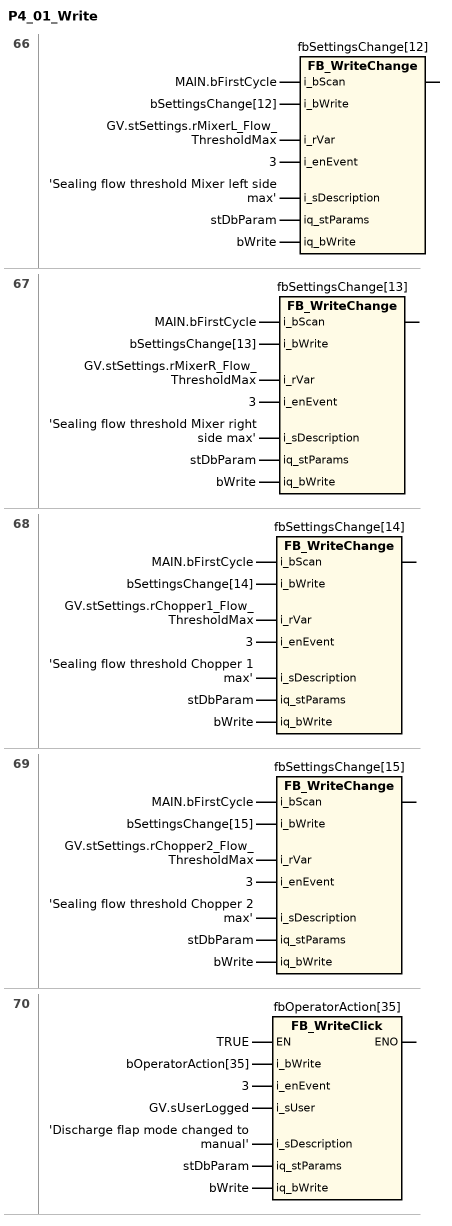
// NETWORK 66
fbSettingsChange[12](
    i_bScan := MAIN.bFirstCycle,
    i_bWrite := bSettingsChange[12],
    i_rVar := GV.stSettings.rMixerL_Flow_ThresholdMax,
    i_enEvent := 3,
    i_sDescription := 'Sealing flow threshold Mixer left side max',
    iq_stParams := stDbParam,
    iq_bWrite := bWrite); // FB_WriteChange

// NETWORK 67
fbSettingsChange[13](
    i_bScan := MAIN.bFirstCycle,
    i_bWrite := bSettingsChange[13],
    i_rVar := GV.stSettings.rMixerR_Flow_ThresholdMax,
    i_enEvent := 3,
    i_sDescription := 'Sealing flow threshold Mixer right side max',
    iq_stParams := stDbParam,
    iq_bWrite := bWrite); // FB_WriteChange

// NETWORK 68
fbSettingsChange[14](
    i_bScan := MAIN.bFirstCycle,
    i_bWrite := bSettingsChange[14],
    i_rVar := GV.stSettings.rChopper1_Flow_ThresholdMax,
    i_enEvent := 3,
    i_sDescription := 'Sealing flow threshold Chopper 1 max',
    iq_stParams := stDbParam,
    iq_bWrite := bWrite); // FB_WriteChange

// NETWORK 69
fbSettingsChange[15](
    i_bScan := MAIN.bFirstCycle,
    i_bWrite := bSettingsChange[15],
    i_rVar := GV.stSettings.rChopper2_Flow_ThresholdMax,
    i_enEvent := 3,
    i_sDescription := 'Sealing flow threshold Chopper 2 max',
    iq_stParams := stDbParam,
    iq_bWrite := bWrite); // FB_WriteChange

// NETWORK 70
fbOperatorAction[35](
    i_bWrite := bOperatorAction[35],
    i_enEvent := 3,
    i_sUser := GV.sUserLogged,
    i_sDescription := 'Discharge flap mode changed to manual',
    iq_stParams := stDbParam,
    iq_bWrite := bWrite); // FB_WriteClick

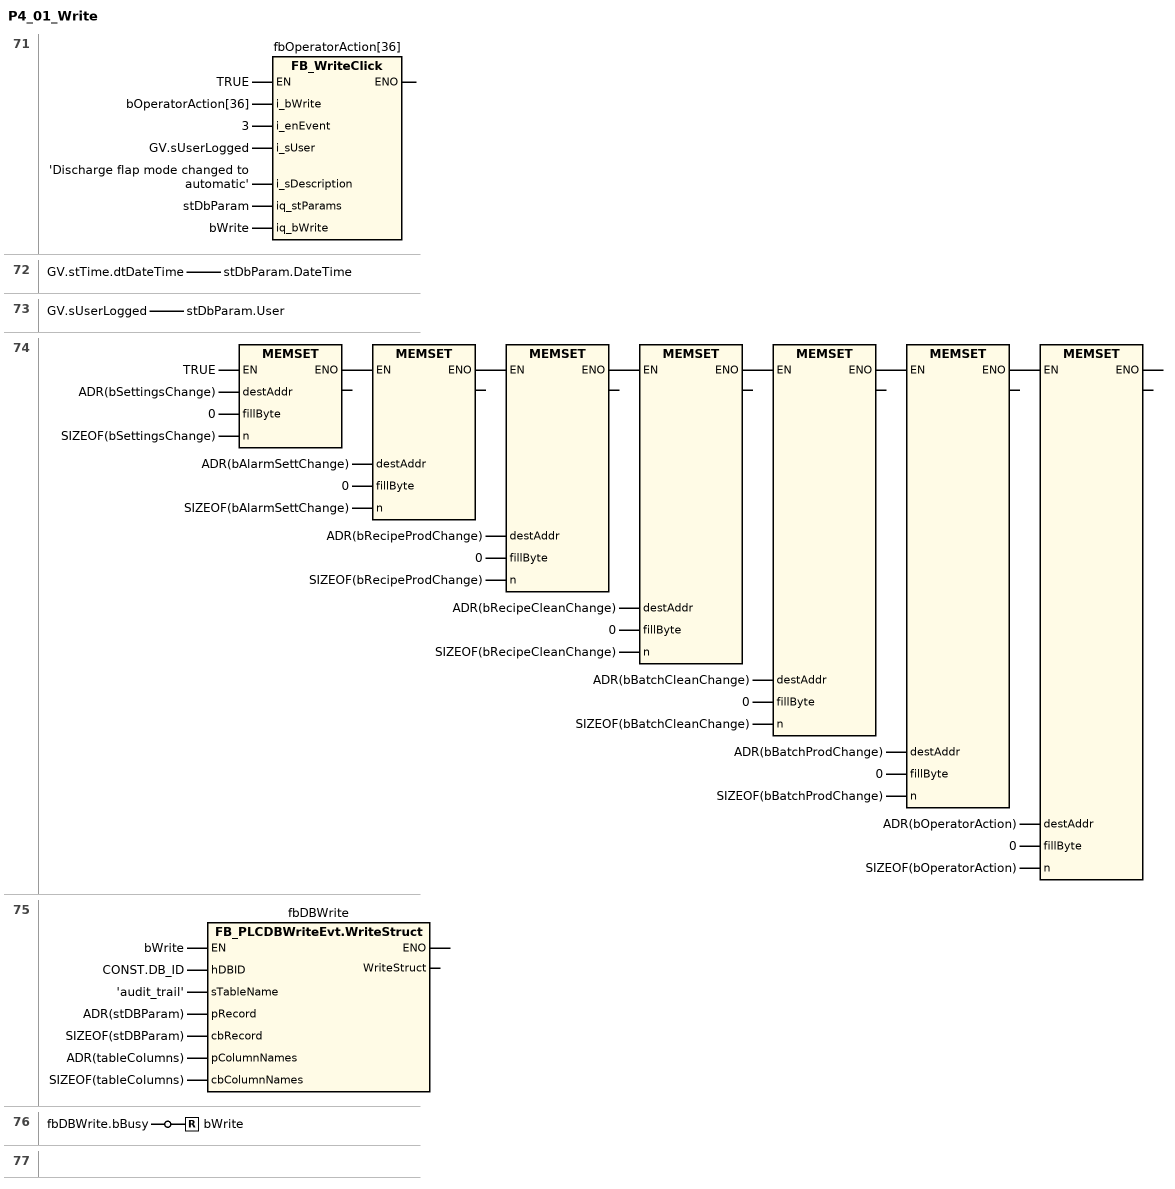
// NETWORK 71
fbOperatorAction[36](
    i_bWrite := bOperatorAction[36],
    i_enEvent := 3,
    i_sUser := GV.sUserLogged,
    i_sDescription := 'Discharge flap mode changed to automatic',
    iq_stParams := stDbParam,
    iq_bWrite := bWrite); // FB_WriteClick

// NETWORK 72
stDbParam.DateTime := GV.stTime.dtDateTime;

// NETWORK 73
stDbParam.User := GV.sUserLogged;

// NETWORK 74
MEMSET(destAddr := ADR(bSettingsChange), fillByte := 0, n := SIZEOF(bSettingsChange));
MEMSET(destAddr := ADR(bAlarmSettChange), fillByte := 0, n := SIZEOF(bAlarmSettChange));
MEMSET(destAddr := ADR(bRecipeProdChange), fillByte := 0, n := SIZEOF(bRecipeProdChange));
MEMSET(destAddr := ADR(bRecipeCleanChange), fillByte := 0, n := SIZEOF(bRecipeCleanChange));
MEMSET(destAddr := ADR(bBatchCleanChange), fillByte := 0, n := SIZEOF(bBatchCleanChange));
MEMSET(destAddr := ADR(bBatchProdChange), fillByte := 0, n := SIZEOF(bBatchProdChange));
MEMSET(destAddr := ADR(bOperatorAction), fillByte := 0, n := SIZEOF(bOperatorAction));

// NETWORK 75
IF bWrite THEN
    fbDBWrite.WriteStruct(
        hDBID := CONST.DB_ID,
        sTableName := 'audit_trail',
        pRecord := ADR(stDBParam),
        cbRecord := SIZEOF(stDBParam),
        pColumnNames := ADR(tableColumns),
        cbColumnNames := SIZEOF(tableColumns));
END_IF

// NETWORK 76
bWrite R= NOT fbDBWrite.bBusy;

// NETWORK 77

END_PROGRAM

// ---- FB/Database/FB_WriteChange.TcPOU
FUNCTION_BLOCK FB_WriteChange
VAR_INPUT
	i_bScan			:BOOL;
	i_bWrite		:BOOL;
	i_rVar			:REAL;
	i_enEvent		:EN_BatchEvents;
	i_sDescription	:STRING;
END_VAR
VAR
	iVarOld			:REAL;
	bVarOld			:BOOL;
	Trig			:R_TRIG;
	bScan			:BOOL;
	Scan			:R_TRIG;
	Scan_TON		:TON;
END_VAR
VAR_IN_OUT
	iq_stParams		:ST_AuditTrail;
	iq_bWrite		:BOOL;
END_VAR

IF i_bScan THEN
	bScan:=TRUE;
END_IF
Scan_TON(IN:=bScan,PT:=T#1S);
IF Scan_TON.Q THEN
	iVarOld:=i_rVar;
	bScan:=FALSE;
END_IF
Trig(CLK:=i_bWrite);
IF Trig.Q AND NOT bScan AND iVarOld <> i_rVar THEN
	iq_stParams.Event:=TO_STRING(i_enEvent);
	iq_stParams.Description := i_sDescription;
	iq_stParams.Oldvalue:=REAL_TO_STRING(iVarOld);
	iq_stParams.Newvalue:=REAL_TO_STRING(i_rVar);
	iVarOld:=i_rVar;
	iq_bWrite:=TRUE;
END_IF

END_FUNCTION_BLOCK

// ---- FB/Database/FB_WriteChange_STR.TcPOU
FUNCTION_BLOCK FB_WriteChange_STR
VAR_INPUT
	i_bScan			:BOOL;
	i_bWrite		:BOOL;
	i_sVar			:STRING;
	i_enEvent		:EN_BatchEvents;
	i_sDescription	:STRING;
END_VAR
VAR
	sVarOld			:STRING;
	bVarOld			:BOOL;
	Trig			:R_TRIG;
	bScan			:BOOL;
	Scan_TON		:TON;
END_VAR
VAR_IN_OUT
	iq_stParams		:ST_AuditTrail;
	iq_bWrite		:BOOL;
END_VAR

IF i_bScan THEN
	bScan:=TRUE;
END_IF
Scan_TON(IN:=bScan,PT:=T#1S);
IF Scan_TON.Q THEN
	sVarOld:=i_sVar;
	bScan:=FALSE;
END_IF
Trig(CLK:=i_bWrite);
IF Trig.Q AND NOT bScan THEN
	iq_stParams.Event:=TO_STRING(i_enEvent);
	iq_stParams.Description := i_sDescription;
	iq_stParams.Oldvalue:=sVarOld;
	iq_stParams.Newvalue:=i_sVar;
	sVarOld:=i_sVar;
	iq_bWrite:=TRUE;
END_IF

END_FUNCTION_BLOCK

// ---- FB/Database/FB_WriteClick.TcPOU
FUNCTION_BLOCK FB_WriteClick
VAR_INPUT
	i_bWrite		:BOOL;
	i_enEvent		:EN_BatchEvents;
	i_sUser			:STRING;
	i_sDescription	:STRING;
END_VAR
VAR
	Trig			:R_TRIG;
END_VAR
VAR_IN_OUT
	iq_stParams		:ST_AuditTrail;
	iq_bWrite		:BOOL;
END_VAR

(*Trig(CLK:=i_bWrite);
IF Trig.Q THEN
	iq_stParams.Event:=TO_STRING(i_enEvent);
	iq_stParams.Description := i_sDescription;
	iq_stParams.Oldvalue:='/';
	iq_stParams.Newvalue:='/';
	iq_bWrite:=TRUE;
END_IF
*)
IF i_bWrite THEN
	iq_stParams.Event:=TO_STRING(i_enEvent);
	iq_stParams.Description := i_sDescription;
	iq_stParams.Oldvalue:='/';
	iq_stParams.Newvalue:='/';
	iq_bWrite:=TRUE;
END_IF

END_FUNCTION_BLOCK

// ---- POUs/4. Audit Trail/P4_02_Read.TcPOU
PROGRAM P4_02_Read
VAR
	fbDBRead    	:FB_PLCDBCmdEvt(sNetID:=CONST.AMS_NETID, tTimeout:=DEFAULT_ADS_TIMEOUT);
	
	tableColumns	:ARRAY [0..5] OF STRING(50) := ['DateTime', 'User', 'Event', 'Description', 'OldValue', 'NewValue'];
	arrParam		:ARRAY [0..5] OF ST_ExpParameter := [(sParaName := 'DateTime', nParaSize := 4, eParaType := E_EXPPARAMETERTYPE.DateTime), 
														(sParaName := 'User', nParaSize := 101, eParaType := E_EXPPARAMETERTYPE.STRING_), 
														(sParaName := 'Event', nParaSize := 101, eParaType := E_EXPPARAMETERTYPE.STRING_), 
														(sParaName := 'Description', nParaSize := 101, eParaType := E_EXPPARAMETERTYPE.STRING_), 
														(sParaName := 'OldValue', nParaSize := 101, eParaType := E_EXPPARAMETERTYPE.STRING_), 
														(sParaName := 'NewValue', nParaSize := 101, eParaType := E_EXPPARAMETERTYPE.STRING_)];
	stRecord		:ARRAY[0..999] OF ST_AuditTrail;	
	
	stDBParam 		:ST_AuditTrail;	
	nRecords		:UDINT;
	sCmd			:STRING[300];

END_VAR
VAR // added by the converter: edge detectors and wires of the graphical bodies
    _w1 : BOOL;
END_VAR

//**************HMI FILTER - COMPOSE QUERY***************
sCmd:='SELECT * FROM `audit_trail`';
IF GV.stHMI.stAudit_Ctrl.bFilter THEN
	
	IF GV.stHMI.stAudit_Ctrl.enFilter_Event <> 0 THEN
		sCmd:=CONCAT(sCmd,'WHERE `Event` = $'');
		sCmd:=CONCAT(sCmD,TO_STRING(GV.stHMI.stAudit_Ctrl.enFilter_Event));
		sCmd:=CONCAT(sCmd,'$'');
	END_IF
	IF GV.stHMI.stAudit_Ctrl.sFilter_User <> GV.sEmptyString THEN
		IF GV.stHMI.stAudit_Ctrl.enFilter_Event = 0 THEN
			sCmd:=CONCAT(sCmd,'WHERE `User` LIKE $'%');
		ELSE
			sCmd:=CONCAT(sCmd,'AND `User` LIKE $'%');
		END_IF
		sCmd:=CONCAT(sCmD,GV.stHMI.stAudit_Ctrl.sFilter_User);
		sCmd:=CONCAT(sCmd,'$'');
	END_IF
	IF GV.stHMI.stAudit_Ctrl.sFilter_Key <> GV.sEmptyString THEN
		IF GV.stHMI.stAudit_Ctrl.enFilter_Event = 0 AND GV.stHMI.stAudit_Ctrl.sFilter_User = GV.sEmptyString THEN
			sCmd:=CONCAT(sCmd,'WHERE `Description` LIKE $'%');
		ELSE
			sCmd:=CONCAT(sCmd,'AND `Description` LIKE $'%');
		END_IF
		sCmd:=CONCAT(sCmD,GV.stHMI.stAudit_Ctrl.sFilter_Key);
		sCmd:=CONCAT(sCmd,'%$'');
	END_IF
	IF GV.stHMI.stAudit_Ctrl.dtFilter_From <> GV.stHMI.stAudit_Ctrl.dtFilter_To THEN
		IF GV.stHMI.stAudit_Ctrl.enFilter_Event = 0 AND GV.stHMI.stAudit_Ctrl.sFilter_User = GV.sEmptyString AND GV.stHMI.stAudit_Ctrl.sFilter_Key = GV.sEmptyString THEN
				sCmd:=CONCAT(sCmd,'WHERE `DateTime` BETWEEN $'');
			ELSE
				sCmd:=CONCAT(sCmd,'AND `DateTime` BETWEEN $'');
			END_IF
			sCmd:=CONCAT(sCmd,RIGHT(DT_TO_STRING(GV.stHMI.stAudit_Ctrl.dtFilter_From),19));
			sCmd:=CONCAT(sCmd,'$' AND $'');
			sCmd:=CONCAT(sCmd,RIGHT(DT_TO_STRING(GV.stHMI.stAudit_Ctrl.dtFilter_To),19));
			sCmd:=CONCAT(sCmd,'$'');
	END_IF
	GV.stTX_Python.sAuditExportQuery:=sCmd;
END_IF
sCmd:=CONCAT(sCmd,' ORDER BY `DateTime` DESC');


ACT_Cmd();

ACTION ACT_Cmd:
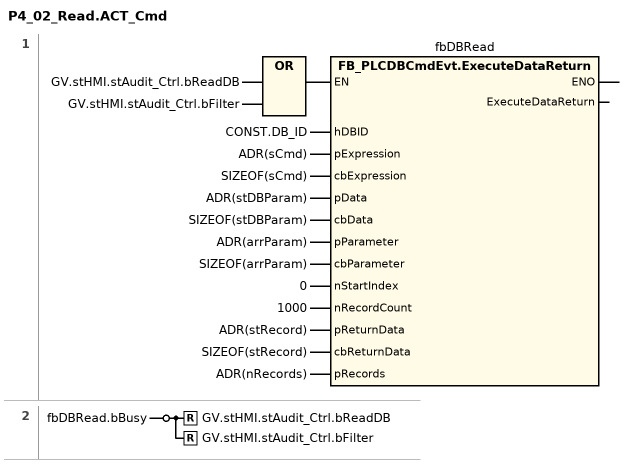
// NETWORK 1
IF GV.stHMI.stAudit_Ctrl.bReadDB OR GV.stHMI.stAudit_Ctrl.bFilter THEN
    fbDBRead.ExecuteDataReturn(
        hDBID := CONST.DB_ID,
        pExpression := ADR(sCmd),
        cbExpression := SIZEOF(sCmd),
        pData := ADR(stDBParam),
        cbData := SIZEOF(stDBParam),
        pParameter := ADR(arrParam),
        cbParameter := SIZEOF(arrParam),
        nStartIndex := 0,
        nRecordCount := 1000,
        pReturnData := ADR(stRecord),
        cbReturnData := SIZEOF(stRecord),
        pRecords := ADR(nRecords));
END_IF

// NETWORK 2
_w1 := NOT fbDBRead.bBusy;
GV.stHMI.stAudit_Ctrl.bReadDB R= _w1;
GV.stHMI.stAudit_Ctrl.bFilter R= _w1;
END_ACTION

END_PROGRAM

// ---- POUs/4. Audit Trail/P4_03_Export.TcPOU
PROGRAM P4_03_Export
VAR
	fbExportAudit					:FB_PythonScript;
END_VAR

VAR PERSISTENT
	sLastExportedAuditTime			:STRING;
	sLastExportedAuditName			:STRING;
END_VAR
VAR // added by the converter: edge detectors and wires of the graphical bodies
    _rt1, _rt2 : R_TRIG;
END_VAR

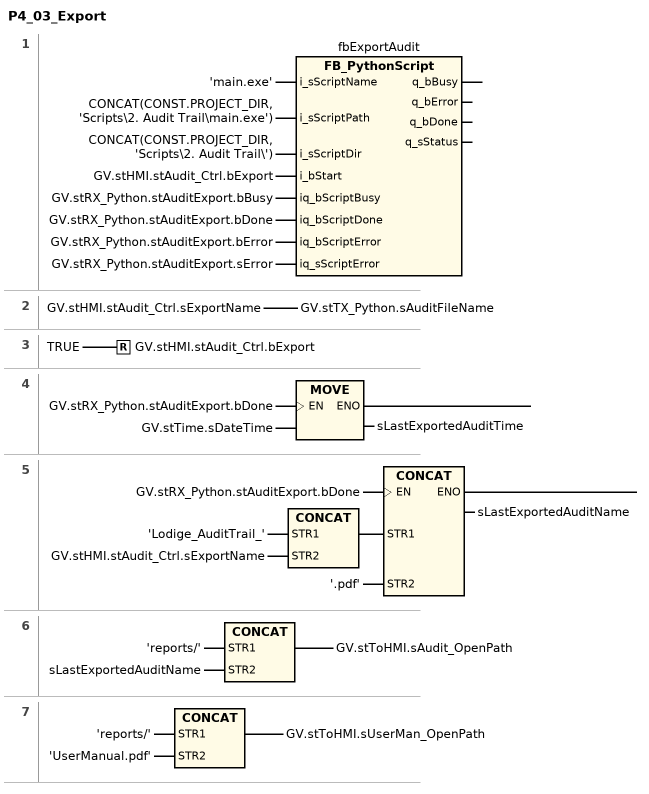
// NETWORK 1
fbExportAudit(
    i_sScriptName := 'main.exe',
    i_sScriptPath := CONCAT(CONST.PROJECT_DIR,'Scripts\2. Audit Trail\main.exe'),
    i_sScriptDir := CONCAT(CONST.PROJECT_DIR,'Scripts\2. Audit Trail\'),
    i_bStart := GV.stHMI.stAudit_Ctrl.bExport,
    iq_bScriptBusy := GV.stRX_Python.stAuditExport.bBusy,
    iq_bScriptDone := GV.stRX_Python.stAuditExport.bDone,
    iq_bScriptError := GV.stRX_Python.stAuditExport.bError,
    iq_sScriptError := GV.stRX_Python.stAuditExport.sError); // FB_PythonScript

// NETWORK 2
GV.stTX_Python.sAuditFileName := GV.stHMI.stAudit_Ctrl.sExportName;

// NETWORK 3
GV.stHMI.stAudit_Ctrl.bExport R= TRUE;

// NETWORK 4
_rt1(CLK := GV.stRX_Python.stAuditExport.bDone);
IF _rt1.Q THEN sLastExportedAuditTime := GV.stTime.sDateTime; END_IF

// NETWORK 5
_rt2(CLK := GV.stRX_Python.stAuditExport.bDone);
IF _rt2.Q THEN
    sLastExportedAuditName := CONCAT(STR1 := CONCAT(STR1 := 'Lodige_AuditTrail_', STR2 := GV.stHMI.stAudit_Ctrl.sExportName), STR2 := '.pdf');
END_IF

// NETWORK 6
GV.stToHMI.sAudit_OpenPath := CONCAT(STR1 := 'reports/', STR2 := sLastExportedAuditName);

// NETWORK 7
GV.stToHMI.sUserMan_OpenPath := CONCAT(STR1 := 'reports/', STR2 := 'UserManual.pdf');

END_PROGRAM

// ---- POUs/4. Audit Trail/P4_04_Delete.TcPOU
PROGRAM P4_04_Delete
VAR
	fbPLCDBCmd    	:FB_PLCDBCmdEvt(sNetID:=CONST.AMS_NETID, tTimeout:=DEFAULT_ADS_TIMEOUT);
	sCmdDelete		:STRING[80];
	
	arrParam		:ARRAY [0..5] OF ST_ExpParameter := [(sParaName := 'DateTime', nParaSize := 4, eParaType := E_EXPPARAMETERTYPE.DateTime), 
														(sParaName := 'User', nParaSize := 101, eParaType := E_EXPPARAMETERTYPE.STRING_), 
														(sParaName := 'Event', nParaSize := 101, eParaType := E_EXPPARAMETERTYPE.STRING_), 
														(sParaName := 'Description', nParaSize := 101, eParaType := E_EXPPARAMETERTYPE.STRING_), 
														(sParaName := 'OldValue', nParaSize := 101, eParaType := E_EXPPARAMETERTYPE.STRING_), 
														(sParaName := 'NewValue', nParaSize := 101, eParaType := E_EXPPARAMETERTYPE.STRING_)];
	
	stDBParam 		:ST_AuditTrail;	
END_VAR

sCmdDelete:='DELETE FROM `audit_trail`';
ACT_Cmd();

ACTION ACT_Cmd:
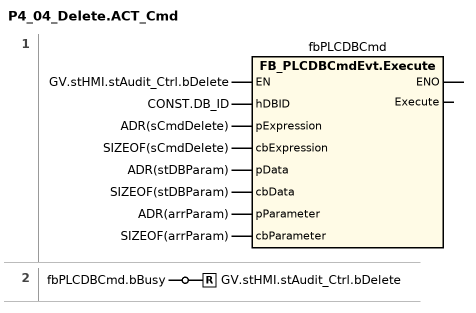
// NETWORK 1
IF GV.stHMI.stAudit_Ctrl.bDelete THEN
    fbPLCDBCmd.Execute(
        hDBID := CONST.DB_ID,
        pExpression := ADR(sCmdDelete),
        cbExpression := SIZEOF(sCmdDelete),
        pData := ADR(stDBParam),
        cbData := SIZEOF(stDBParam),
        pParameter := ADR(arrParam),
        cbParameter := SIZEOF(arrParam));
END_IF

// NETWORK 2
GV.stHMI.stAudit_Ctrl.bDelete R= NOT fbPLCDBCmd.bBusy;
END_ACTION

END_PROGRAM

// ---- POUs/4. Audit Trail/P4_05_Send.TcPOU
PROGRAM P4_05_Send
VAR
	fbAuditSend							:FB_PythonScript;
END_VAR
VAR // added by the converter: edge detectors and wires of the graphical bodies
    _rt1 : R_TRIG;
END_VAR

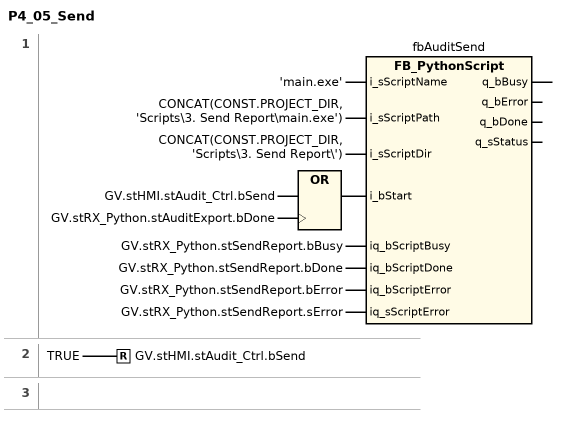
// NETWORK 1
_rt1(CLK := GV.stRX_Python.stAuditExport.bDone);
fbAuditSend(
    i_sScriptName := 'main.exe',
    i_sScriptPath := CONCAT(CONST.PROJECT_DIR,'Scripts\3. Send Report\main.exe'),
    i_sScriptDir := CONCAT(CONST.PROJECT_DIR,'Scripts\3. Send Report\'),
    i_bStart := GV.stHMI.stAudit_Ctrl.bSend OR _rt1.Q,
    iq_bScriptBusy := GV.stRX_Python.stSendReport.bBusy,
    iq_bScriptDone := GV.stRX_Python.stSendReport.bDone,
    iq_bScriptError := GV.stRX_Python.stSendReport.bError,
    iq_sScriptError := GV.stRX_Python.stSendReport.sError); // FB_PythonScript

// NETWORK 2
GV.stHMI.stAudit_Ctrl.bSend R= TRUE;

// NETWORK 3

END_PROGRAM

// ---- POUs/4. Audit Trail/P4_05_DIskSize.TcPOU
PROGRAM P4_05_DIskSize
VAR
	fbSize				:FB_PythonScript;
END_VAR

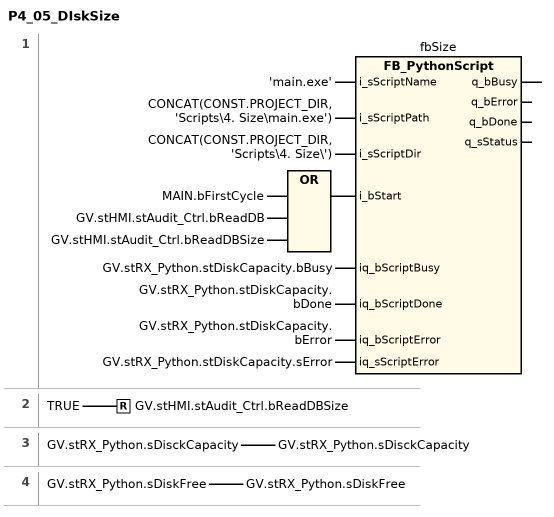
// NETWORK 1
fbSize(
    i_sScriptName := 'main.exe',
    i_sScriptPath := CONCAT(CONST.PROJECT_DIR,'Scripts\4. Size\main.exe'),
    i_sScriptDir := CONCAT(CONST.PROJECT_DIR,'Scripts\4. Size\'),
    i_bStart := MAIN.bFirstCycle OR GV.stHMI.stAudit_Ctrl.bReadDB OR GV.stHMI.stAudit_Ctrl.bReadDBSize,
    iq_bScriptBusy := GV.stRX_Python.stDiskCapacity.bBusy,
    iq_bScriptDone := GV.stRX_Python.stDiskCapacity.bDone,
    iq_bScriptError := GV.stRX_Python.stDiskCapacity.bError,
    iq_sScriptError := GV.stRX_Python.stDiskCapacity.sError); // FB_PythonScript

// NETWORK 2
GV.stHMI.stAudit_Ctrl.bReadDBSize R= TRUE;

// NETWORK 3
GV.stRX_Python.sDisckCapacity := GV.stRX_Python.sDisckCapacity;

// NETWORK 4
GV.stRX_Python.sDiskFree := GV.stRX_Python.sDiskFree;

END_PROGRAM

// ---- POUs/5. HMI/P5_00_MAIN.TcPOU
PROGRAM P5_00_MAIN
VAR

END_VAR

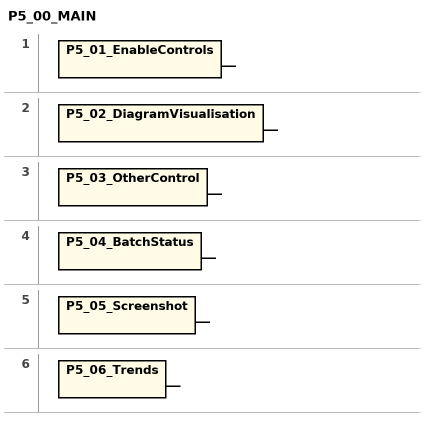
// NETWORK 1
P5_01_EnableControls();

// NETWORK 2
P5_02_DiagramVisualisation();

// NETWORK 3
P5_03_OtherControl();

// NETWORK 4
P5_04_BatchStatus();

// NETWORK 5
P5_05_Screenshot();

// NETWORK 6
P5_06_Trends();

END_PROGRAM

// ---- POUs/5. HMI/P5_01_EnableControls.TcPOU
PROGRAM P5_01_EnableControls
VAR
	tonDisableNext			:TON;
	tonDisablePrev			:TON;
END_VAR
VAR // added by the converter: edge detectors and wires of the graphical bodies
    _w1, _w2 : BOOL;
END_VAR

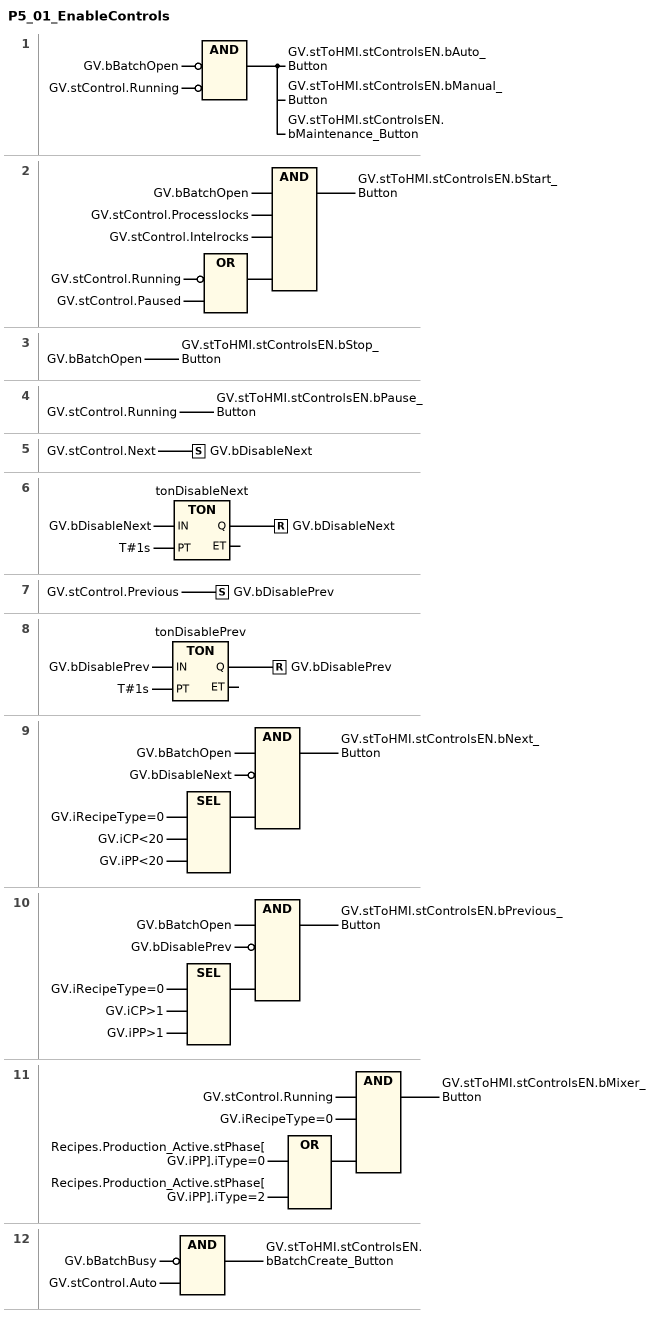
// NETWORK 1
_w1 := NOT GV.bBatchOpen AND NOT GV.stControl.Running;
GV.stToHMI.stControlsEN.bAuto_Button := _w1;
GV.stToHMI.stControlsEN.bManual_Button := _w1;
GV.stToHMI.stControlsEN.bMaintenance_Button := _w1;

// NETWORK 2
GV.stToHMI.stControlsEN.bStart_Button := GV.bBatchOpen AND GV.stControl.Processlocks AND GV.stControl.Intelrocks AND (NOT GV.stControl.Running OR GV.stControl.Paused);

// NETWORK 3
GV.stToHMI.stControlsEN.bStop_Button := GV.bBatchOpen;

// NETWORK 4
GV.stToHMI.stControlsEN.bPause_Button := GV.stControl.Running;

// NETWORK 5
GV.bDisableNext S= GV.stControl.Next;

// NETWORK 6
tonDisableNext(IN := GV.bDisableNext, PT := T#1s); // TON
GV.bDisableNext R= tonDisableNext.Q;

// NETWORK 7
GV.bDisablePrev S= GV.stControl.Previous;

// NETWORK 8
tonDisablePrev(IN := GV.bDisablePrev, PT := T#1s); // TON
GV.bDisablePrev R= tonDisablePrev.Q;

// NETWORK 9
GV.stToHMI.stControlsEN.bNext_Button := GV.bBatchOpen AND NOT GV.bDisableNext AND SEL(GV.iRecipeType=0, GV.iCP<20, GV.iPP<20);

// NETWORK 10
GV.stToHMI.stControlsEN.bPrevious_Button := GV.bBatchOpen AND NOT GV.bDisablePrev AND SEL(GV.iRecipeType=0, GV.iCP>1, GV.iPP>1);

// NETWORK 11
GV.stToHMI.stControlsEN.bMixer_Button := GV.stControl.Running AND (GV.iRecipeType=0) AND ((Recipes.Production_Active.stPhase[GV.iPP].iType=0) OR (Recipes.Production_Active.stPhase[GV.iPP].iType=2));

// NETWORK 12
GV.stToHMI.stControlsEN.bBatchCreate_Button := NOT GV.bBatchBusy AND GV.stControl.Auto;

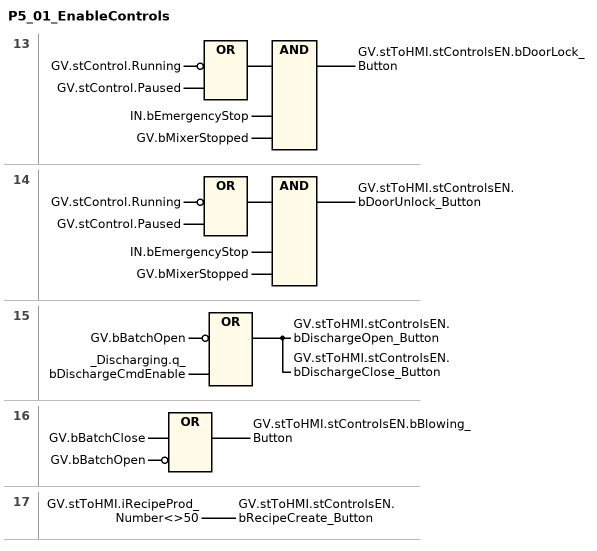
// NETWORK 13
GV.stToHMI.stControlsEN.bDoorLock_Button := (NOT GV.stControl.Running OR GV.stControl.Paused) AND IN.bEmergencyStop AND GV.bMixerStopped;

// NETWORK 14
GV.stToHMI.stControlsEN.bDoorUnlock_Button := (NOT GV.stControl.Running OR GV.stControl.Paused) AND IN.bEmergencyStop AND GV.bMixerStopped;

// NETWORK 15
_w2 := NOT GV.bBatchOpen OR _Discharging.q_bDischargeCmdEnable;
GV.stToHMI.stControlsEN.bDischargeOpen_Button := _w2;
GV.stToHMI.stControlsEN.bDischargeClose_Button := _w2;

// NETWORK 16
GV.stToHMI.stControlsEN.bBlowing_Button := GV.bBatchClose OR NOT GV.bBatchOpen;

// NETWORK 17
GV.stToHMI.stControlsEN.bRecipeCreate_Button := GV.stToHMI.iRecipeProd_Number<>50;

END_PROGRAM

// ---- POUs/5. HMI/P5_02_DiagramVisualisation.TcPOU
PROGRAM P5_02_DiagramVisualisation
VAR
END_VAR

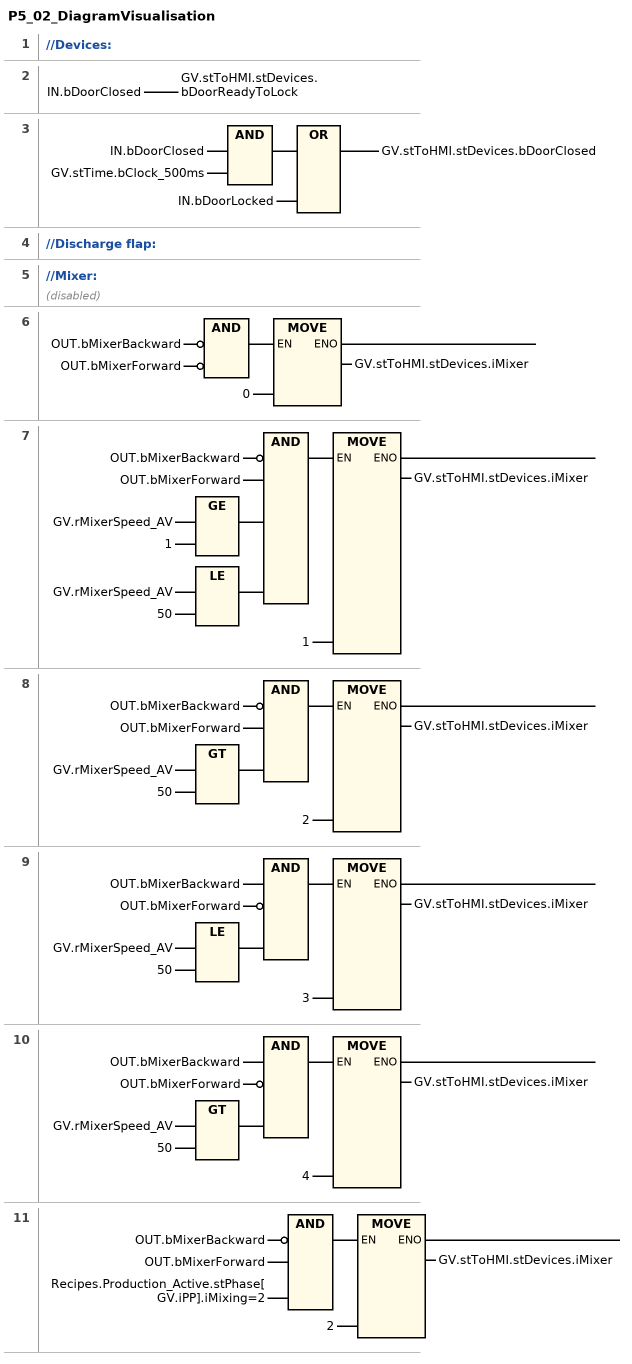
// NETWORK 1
// label: //Devices

// NETWORK 2
GV.stToHMI.stDevices.bDoorReadyToLock := IN.bDoorClosed;

// NETWORK 3
GV.stToHMI.stDevices.bDoorClosed := IN.bDoorClosed AND GV.stTime.bClock_500ms OR IN.bDoorLocked;

// NETWORK 4
// label: //Discharge flap

// NETWORK 5 (disabled)
// label: //Mixer

// NETWORK 6
IF NOT OUT.bMixerBackward AND NOT OUT.bMixerForward THEN GV.stToHMI.stDevices.iMixer := 0; END_IF

// NETWORK 7
IF NOT OUT.bMixerBackward AND OUT.bMixerForward AND GV.rMixerSpeed_AV >= 1 AND GV.rMixerSpeed_AV <= 50 THEN
    GV.stToHMI.stDevices.iMixer := 1;
END_IF

// NETWORK 8
IF NOT OUT.bMixerBackward AND OUT.bMixerForward AND GV.rMixerSpeed_AV > 50 THEN
    GV.stToHMI.stDevices.iMixer := 2;
END_IF

// NETWORK 9
IF OUT.bMixerBackward AND NOT OUT.bMixerForward AND GV.rMixerSpeed_AV <= 50 THEN
    GV.stToHMI.stDevices.iMixer := 3;
END_IF

// NETWORK 10
IF OUT.bMixerBackward AND NOT OUT.bMixerForward AND GV.rMixerSpeed_AV > 50 THEN
    GV.stToHMI.stDevices.iMixer := 4;
END_IF

// NETWORK 11
IF NOT OUT.bMixerBackward AND OUT.bMixerForward AND (Recipes.Production_Active.stPhase[GV.iPP].iMixing=2) THEN
    GV.stToHMI.stDevices.iMixer := 2;
END_IF

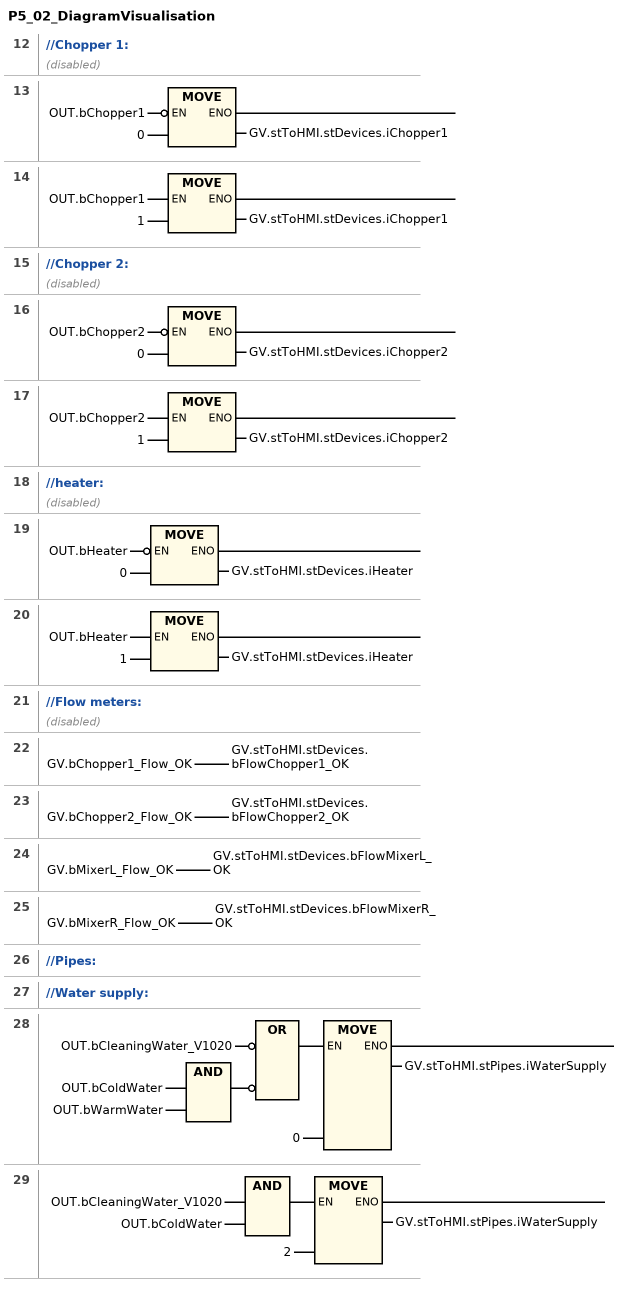
// NETWORK 12 (disabled)
// label: //Chopper 1

// NETWORK 13
IF NOT OUT.bChopper1 THEN GV.stToHMI.stDevices.iChopper1 := 0; END_IF

// NETWORK 14
IF OUT.bChopper1 THEN GV.stToHMI.stDevices.iChopper1 := 1; END_IF

// NETWORK 15 (disabled)
// label: //Chopper 2

// NETWORK 16
IF NOT OUT.bChopper2 THEN GV.stToHMI.stDevices.iChopper2 := 0; END_IF

// NETWORK 17
IF OUT.bChopper2 THEN GV.stToHMI.stDevices.iChopper2 := 1; END_IF

// NETWORK 18 (disabled)
// label: //heater

// NETWORK 19
IF NOT OUT.bHeater THEN GV.stToHMI.stDevices.iHeater := 0; END_IF

// NETWORK 20
IF OUT.bHeater THEN GV.stToHMI.stDevices.iHeater := 1; END_IF

// NETWORK 21 (disabled)
// label: //Flow meters

// NETWORK 22
GV.stToHMI.stDevices.bFlowChopper1_OK := GV.bChopper1_Flow_OK;

// NETWORK 23
GV.stToHMI.stDevices.bFlowChopper2_OK := GV.bChopper2_Flow_OK;

// NETWORK 24
GV.stToHMI.stDevices.bFlowMixerL_OK := GV.bMixerL_Flow_OK;

// NETWORK 25
GV.stToHMI.stDevices.bFlowMixerR_OK := GV.bMixerR_Flow_OK;

// NETWORK 26
// label: //Pipes

// NETWORK 27
// label: //Water supply

// NETWORK 28
IF NOT OUT.bCleaningWater_V1020 OR NOT (OUT.bColdWater AND OUT.bWarmWater) THEN
    GV.stToHMI.stPipes.iWaterSupply := 0;
END_IF

// NETWORK 29
IF OUT.bCleaningWater_V1020 AND OUT.bColdWater THEN GV.stToHMI.stPipes.iWaterSupply := 2; END_IF

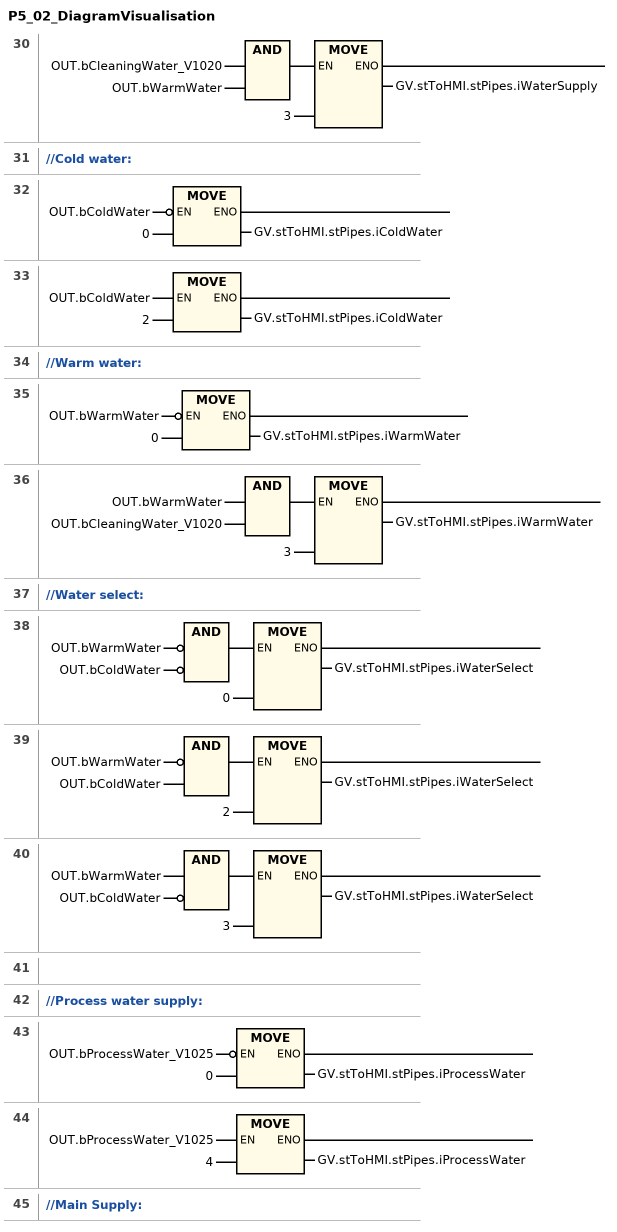
// NETWORK 30
IF OUT.bCleaningWater_V1020 AND OUT.bWarmWater THEN GV.stToHMI.stPipes.iWaterSupply := 3; END_IF

// NETWORK 31
// label: //Cold water

// NETWORK 32
IF NOT OUT.bColdWater THEN GV.stToHMI.stPipes.iColdWater := 0; END_IF

// NETWORK 33
IF OUT.bColdWater THEN GV.stToHMI.stPipes.iColdWater := 2; END_IF

// NETWORK 34
// label: //Warm water

// NETWORK 35
IF NOT OUT.bWarmWater THEN GV.stToHMI.stPipes.iWarmWater := 0; END_IF

// NETWORK 36
IF OUT.bWarmWater AND OUT.bCleaningWater_V1020 THEN GV.stToHMI.stPipes.iWarmWater := 3; END_IF

// NETWORK 37
// label: //Water select

// NETWORK 38
IF NOT OUT.bWarmWater AND NOT OUT.bColdWater THEN GV.stToHMI.stPipes.iWaterSelect := 0; END_IF

// NETWORK 39
IF NOT OUT.bWarmWater AND OUT.bColdWater THEN GV.stToHMI.stPipes.iWaterSelect := 2; END_IF

// NETWORK 40
IF OUT.bWarmWater AND NOT OUT.bColdWater THEN GV.stToHMI.stPipes.iWaterSelect := 3; END_IF

// NETWORK 41

// NETWORK 42
// label: //Process water supply

// NETWORK 43
IF NOT OUT.bProcessWater_V1025 THEN GV.stToHMI.stPipes.iProcessWater := 0; END_IF

// NETWORK 44
IF OUT.bProcessWater_V1025 THEN GV.stToHMI.stPipes.iProcessWater := 4; END_IF

// NETWORK 45
// label: //Main Supply

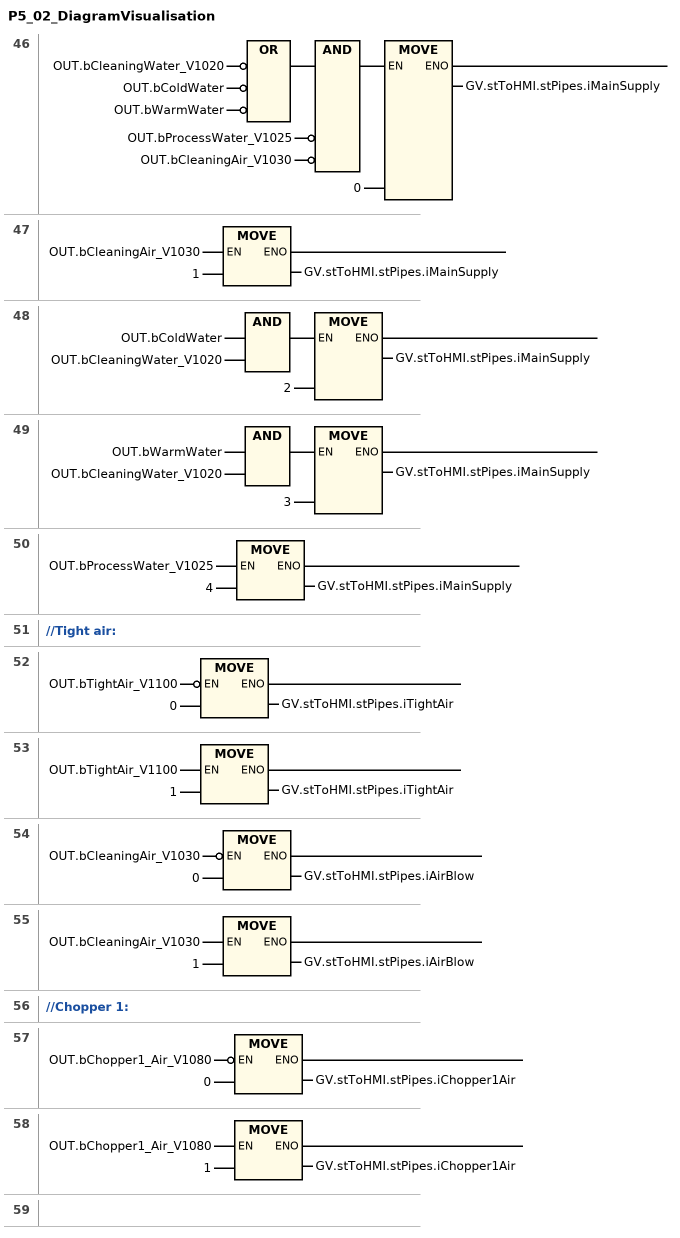
// NETWORK 46
IF (NOT OUT.bCleaningWater_V1020 OR NOT OUT.bColdWater OR NOT OUT.bWarmWater) AND NOT OUT.bProcessWater_V1025 AND NOT OUT.bCleaningAir_V1030 THEN
    GV.stToHMI.stPipes.iMainSupply := 0;
END_IF

// NETWORK 47
IF OUT.bCleaningAir_V1030 THEN GV.stToHMI.stPipes.iMainSupply := 1; END_IF

// NETWORK 48
IF OUT.bColdWater AND OUT.bCleaningWater_V1020 THEN GV.stToHMI.stPipes.iMainSupply := 2; END_IF

// NETWORK 49
IF OUT.bWarmWater AND OUT.bCleaningWater_V1020 THEN GV.stToHMI.stPipes.iMainSupply := 3; END_IF

// NETWORK 50
IF OUT.bProcessWater_V1025 THEN GV.stToHMI.stPipes.iMainSupply := 4; END_IF

// NETWORK 51
// label: //Tight air

// NETWORK 52
IF NOT OUT.bTightAir_V1100 THEN GV.stToHMI.stPipes.iTightAir := 0; END_IF

// NETWORK 53
IF OUT.bTightAir_V1100 THEN GV.stToHMI.stPipes.iTightAir := 1; END_IF

// NETWORK 54
IF NOT OUT.bCleaningAir_V1030 THEN GV.stToHMI.stPipes.iAirBlow := 0; END_IF

// NETWORK 55
IF OUT.bCleaningAir_V1030 THEN GV.stToHMI.stPipes.iAirBlow := 1; END_IF

// NETWORK 56
// label: //Chopper 1

// NETWORK 57
IF NOT OUT.bChopper1_Air_V1080 THEN GV.stToHMI.stPipes.iChopper1Air := 0; END_IF

// NETWORK 58
IF OUT.bChopper1_Air_V1080 THEN GV.stToHMI.stPipes.iChopper1Air := 1; END_IF

// NETWORK 59

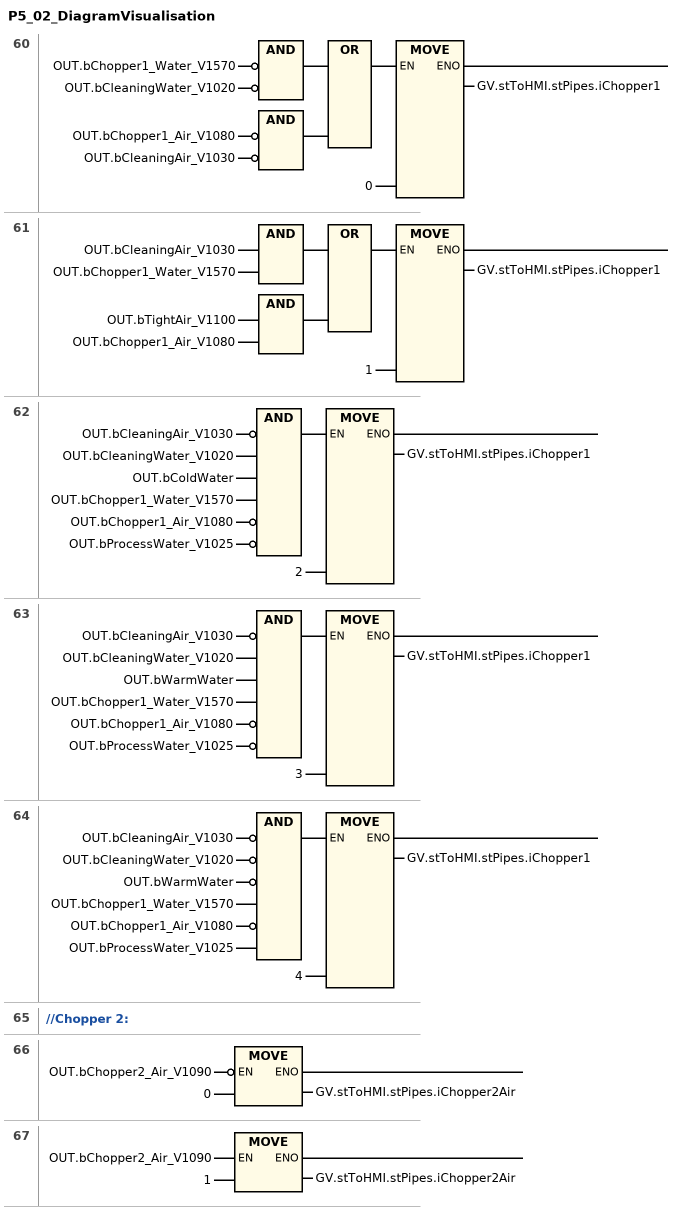
// NETWORK 60
IF NOT OUT.bChopper1_Water_V1570 AND NOT OUT.bCleaningWater_V1020 OR NOT OUT.bChopper1_Air_V1080 AND NOT OUT.bCleaningAir_V1030 THEN
    GV.stToHMI.stPipes.iChopper1 := 0;
END_IF

// NETWORK 61
IF OUT.bCleaningAir_V1030 AND OUT.bChopper1_Water_V1570 OR OUT.bTightAir_V1100 AND OUT.bChopper1_Air_V1080 THEN
    GV.stToHMI.stPipes.iChopper1 := 1;
END_IF

// NETWORK 62
IF NOT OUT.bCleaningAir_V1030 AND OUT.bCleaningWater_V1020 AND OUT.bColdWater AND OUT.bChopper1_Water_V1570 AND NOT OUT.bChopper1_Air_V1080 AND NOT OUT.bProcessWater_V1025 THEN
    GV.stToHMI.stPipes.iChopper1 := 2;
END_IF

// NETWORK 63
IF NOT OUT.bCleaningAir_V1030 AND OUT.bCleaningWater_V1020 AND OUT.bWarmWater AND OUT.bChopper1_Water_V1570 AND NOT OUT.bChopper1_Air_V1080 AND NOT OUT.bProcessWater_V1025 THEN
    GV.stToHMI.stPipes.iChopper1 := 3;
END_IF

// NETWORK 64
IF NOT OUT.bCleaningAir_V1030 AND NOT OUT.bCleaningWater_V1020 AND NOT OUT.bWarmWater AND OUT.bChopper1_Water_V1570 AND NOT OUT.bChopper1_Air_V1080 AND OUT.bProcessWater_V1025 THEN
    GV.stToHMI.stPipes.iChopper1 := 4;
END_IF

// NETWORK 65
// label: //Chopper 2

// NETWORK 66
IF NOT OUT.bChopper2_Air_V1090 THEN GV.stToHMI.stPipes.iChopper2Air := 0; END_IF

// NETWORK 67
IF OUT.bChopper2_Air_V1090 THEN GV.stToHMI.stPipes.iChopper2Air := 1; END_IF

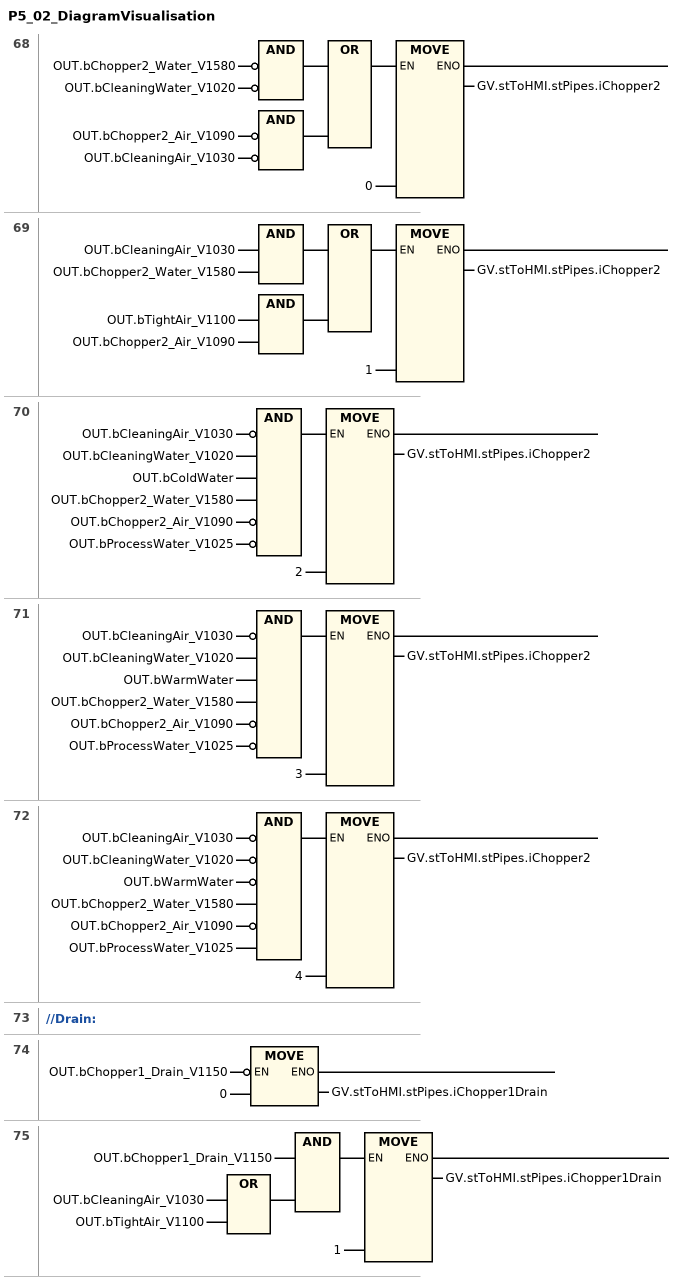
// NETWORK 68
IF NOT OUT.bChopper2_Water_V1580 AND NOT OUT.bCleaningWater_V1020 OR NOT OUT.bChopper2_Air_V1090 AND NOT OUT.bCleaningAir_V1030 THEN
    GV.stToHMI.stPipes.iChopper2 := 0;
END_IF

// NETWORK 69
IF OUT.bCleaningAir_V1030 AND OUT.bChopper2_Water_V1580 OR OUT.bTightAir_V1100 AND OUT.bChopper2_Air_V1090 THEN
    GV.stToHMI.stPipes.iChopper2 := 1;
END_IF

// NETWORK 70
IF NOT OUT.bCleaningAir_V1030 AND OUT.bCleaningWater_V1020 AND OUT.bColdWater AND OUT.bChopper2_Water_V1580 AND NOT OUT.bChopper2_Air_V1090 AND NOT OUT.bProcessWater_V1025 THEN
    GV.stToHMI.stPipes.iChopper2 := 2;
END_IF

// NETWORK 71
IF NOT OUT.bCleaningAir_V1030 AND OUT.bCleaningWater_V1020 AND OUT.bWarmWater AND OUT.bChopper2_Water_V1580 AND NOT OUT.bChopper2_Air_V1090 AND NOT OUT.bProcessWater_V1025 THEN
    GV.stToHMI.stPipes.iChopper2 := 3;
END_IF

// NETWORK 72
IF NOT OUT.bCleaningAir_V1030 AND NOT OUT.bCleaningWater_V1020 AND NOT OUT.bWarmWater AND OUT.bChopper2_Water_V1580 AND NOT OUT.bChopper2_Air_V1090 AND OUT.bProcessWater_V1025 THEN
    GV.stToHMI.stPipes.iChopper2 := 4;
END_IF

// NETWORK 73
// label: //Drain

// NETWORK 74
IF NOT OUT.bChopper1_Drain_V1150 THEN GV.stToHMI.stPipes.iChopper1Drain := 0; END_IF

// NETWORK 75
IF OUT.bChopper1_Drain_V1150 AND (OUT.bCleaningAir_V1030 OR OUT.bTightAir_V1100) THEN
    GV.stToHMI.stPipes.iChopper1Drain := 1;
END_IF

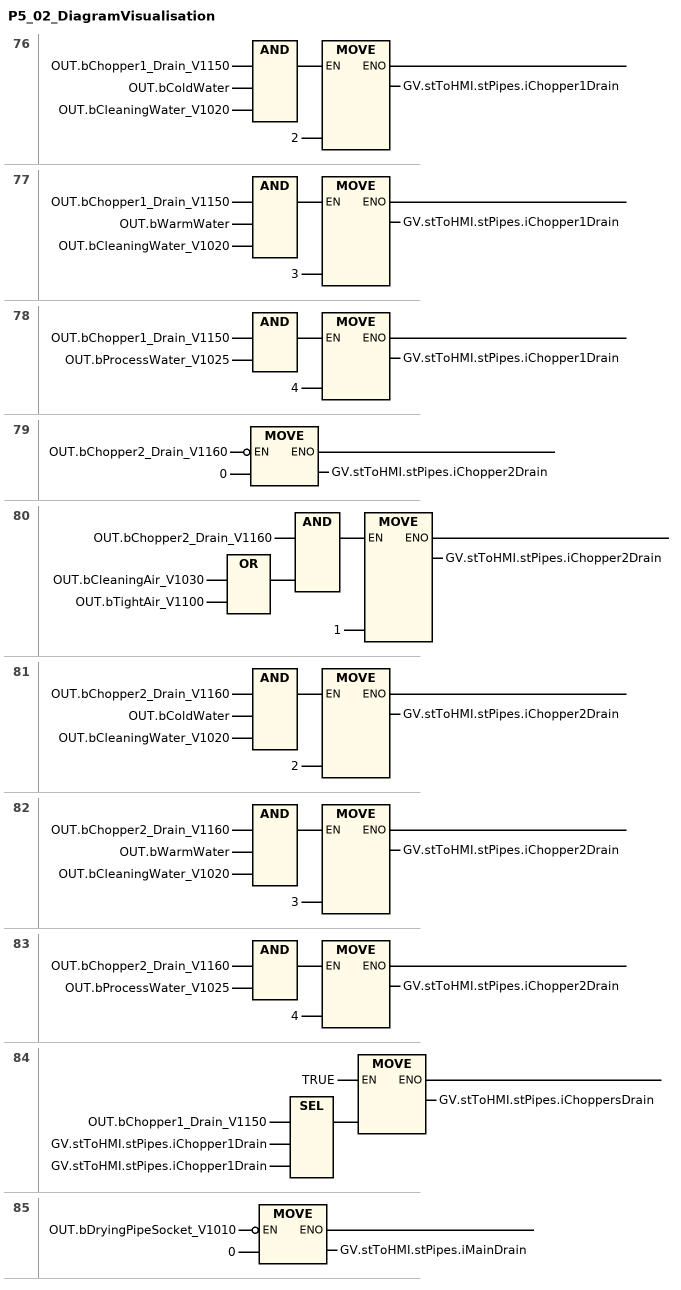
// NETWORK 76
IF OUT.bChopper1_Drain_V1150 AND OUT.bColdWater AND OUT.bCleaningWater_V1020 THEN
    GV.stToHMI.stPipes.iChopper1Drain := 2;
END_IF

// NETWORK 77
IF OUT.bChopper1_Drain_V1150 AND OUT.bWarmWater AND OUT.bCleaningWater_V1020 THEN
    GV.stToHMI.stPipes.iChopper1Drain := 3;
END_IF

// NETWORK 78
IF OUT.bChopper1_Drain_V1150 AND OUT.bProcessWater_V1025 THEN GV.stToHMI.stPipes.iChopper1Drain := 4; END_IF

// NETWORK 79
IF NOT OUT.bChopper2_Drain_V1160 THEN GV.stToHMI.stPipes.iChopper2Drain := 0; END_IF

// NETWORK 80
IF OUT.bChopper2_Drain_V1160 AND (OUT.bCleaningAir_V1030 OR OUT.bTightAir_V1100) THEN
    GV.stToHMI.stPipes.iChopper2Drain := 1;
END_IF

// NETWORK 81
IF OUT.bChopper2_Drain_V1160 AND OUT.bColdWater AND OUT.bCleaningWater_V1020 THEN
    GV.stToHMI.stPipes.iChopper2Drain := 2;
END_IF

// NETWORK 82
IF OUT.bChopper2_Drain_V1160 AND OUT.bWarmWater AND OUT.bCleaningWater_V1020 THEN
    GV.stToHMI.stPipes.iChopper2Drain := 3;
END_IF

// NETWORK 83
IF OUT.bChopper2_Drain_V1160 AND OUT.bProcessWater_V1025 THEN GV.stToHMI.stPipes.iChopper2Drain := 4; END_IF

// NETWORK 84
GV.stToHMI.stPipes.iChoppersDrain := SEL(OUT.bChopper1_Drain_V1150, GV.stToHMI.stPipes.iChopper1Drain, GV.stToHMI.stPipes.iChopper1Drain);

// NETWORK 85
IF NOT OUT.bDryingPipeSocket_V1010 THEN GV.stToHMI.stPipes.iMainDrain := 0; END_IF

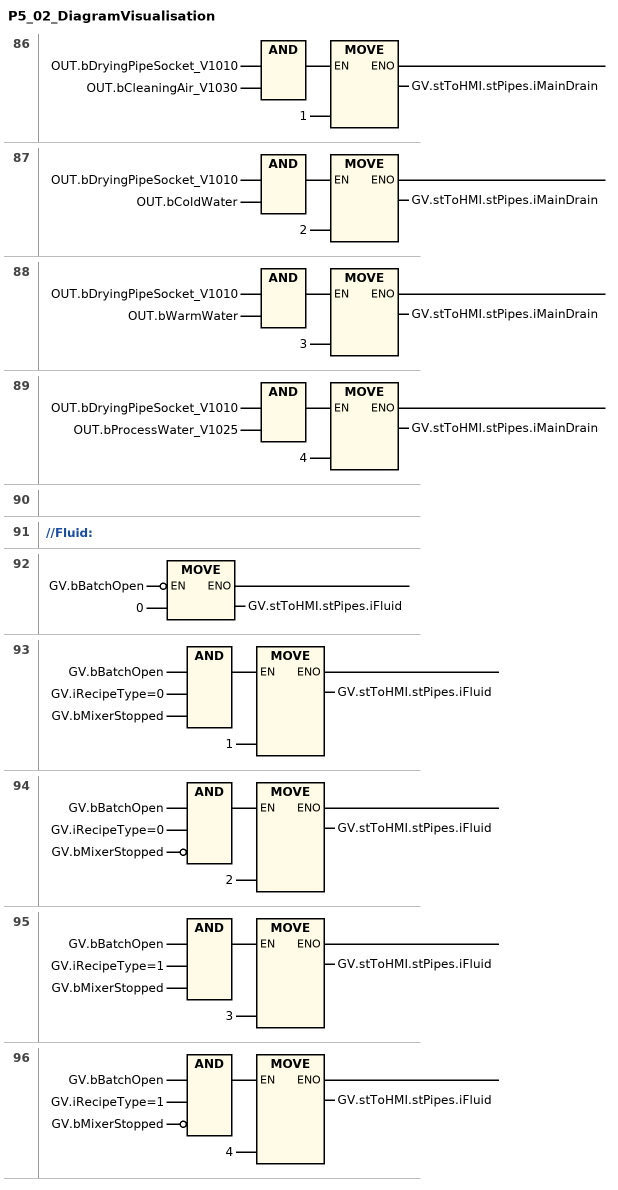
// NETWORK 86
IF OUT.bDryingPipeSocket_V1010 AND OUT.bCleaningAir_V1030 THEN GV.stToHMI.stPipes.iMainDrain := 1; END_IF

// NETWORK 87
IF OUT.bDryingPipeSocket_V1010 AND OUT.bColdWater THEN GV.stToHMI.stPipes.iMainDrain := 2; END_IF

// NETWORK 88
IF OUT.bDryingPipeSocket_V1010 AND OUT.bWarmWater THEN GV.stToHMI.stPipes.iMainDrain := 3; END_IF

// NETWORK 89
IF OUT.bDryingPipeSocket_V1010 AND OUT.bProcessWater_V1025 THEN GV.stToHMI.stPipes.iMainDrain := 4; END_IF

// NETWORK 90

// NETWORK 91
// label: //Fluid

// NETWORK 92
IF NOT GV.bBatchOpen THEN GV.stToHMI.stPipes.iFluid := 0; END_IF

// NETWORK 93
IF GV.bBatchOpen AND (GV.iRecipeType=0) AND GV.bMixerStopped THEN GV.stToHMI.stPipes.iFluid := 1; END_IF

// NETWORK 94
IF GV.bBatchOpen AND (GV.iRecipeType=0) AND NOT GV.bMixerStopped THEN GV.stToHMI.stPipes.iFluid := 2; END_IF

// NETWORK 95
IF GV.bBatchOpen AND (GV.iRecipeType=1) AND GV.bMixerStopped THEN GV.stToHMI.stPipes.iFluid := 3; END_IF

// NETWORK 96
IF GV.bBatchOpen AND (GV.iRecipeType=1) AND NOT GV.bMixerStopped THEN GV.stToHMI.stPipes.iFluid := 4; END_IF

END_PROGRAM

// ---- POUs/5. HMI/P5_03_OtherControl.TcPOU
PROGRAM P5_03_OtherControl
VAR
END_VAR

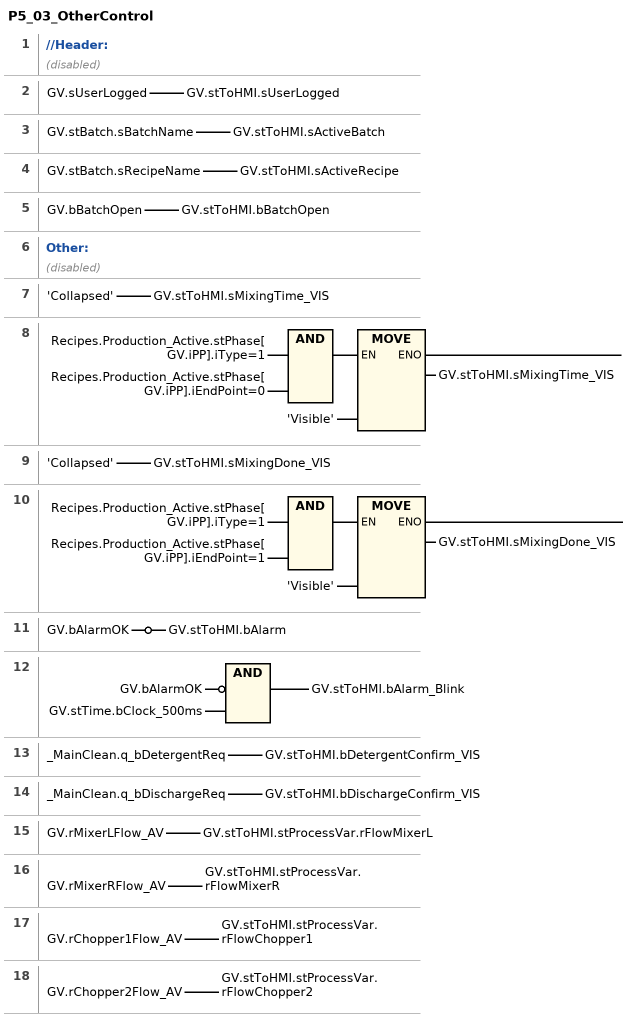
// NETWORK 1 (disabled)
// label: //Header

// NETWORK 2
GV.stToHMI.sUserLogged := GV.sUserLogged;

// NETWORK 3
GV.stToHMI.sActiveBatch := GV.stBatch.sBatchName;

// NETWORK 4
GV.stToHMI.sActiveRecipe := GV.stBatch.sRecipeName;

// NETWORK 5
GV.stToHMI.bBatchOpen := GV.bBatchOpen;

// NETWORK 6 (disabled)
// label: Other

// NETWORK 7
GV.stToHMI.sMixingTime_VIS := 'Collapsed';

// NETWORK 8
IF (Recipes.Production_Active.stPhase[GV.iPP].iType=1) AND (Recipes.Production_Active.stPhase[GV.iPP].iEndPoint=0) THEN
    GV.stToHMI.sMixingTime_VIS := 'Visible';
END_IF

// NETWORK 9
GV.stToHMI.sMixingDone_VIS := 'Collapsed';

// NETWORK 10
IF (Recipes.Production_Active.stPhase[GV.iPP].iType=1) AND (Recipes.Production_Active.stPhase[GV.iPP].iEndPoint=1) THEN
    GV.stToHMI.sMixingDone_VIS := 'Visible';
END_IF

// NETWORK 11
GV.stToHMI.bAlarm := NOT GV.bAlarmOK;

// NETWORK 12
GV.stToHMI.bAlarm_Blink := NOT GV.bAlarmOK AND GV.stTime.bClock_500ms;

// NETWORK 13
GV.stToHMI.bDetergentConfirm_VIS := _MainClean.q_bDetergentReq;

// NETWORK 14
GV.stToHMI.bDischargeConfirm_VIS := _MainClean.q_bDischargeReq;

// NETWORK 15
GV.stToHMI.stProcessVar.rFlowMixerL := GV.rMixerLFlow_AV;

// NETWORK 16
GV.stToHMI.stProcessVar.rFlowMixerR := GV.rMixerRFlow_AV;

// NETWORK 17
GV.stToHMI.stProcessVar.rFlowChopper1 := GV.rChopper1Flow_AV;

// NETWORK 18
GV.stToHMI.stProcessVar.rFlowChopper2 := GV.rChopper2Flow_AV;

END_PROGRAM

// ---- POUs/5. HMI/P5_04_BatchStatus.TcPOU
PROGRAM P5_04_BatchStatus
VAR
	tonBatchOpen			:TON;
	tPhaseTimeET			:TIME;
	tSubStep1Prod			:TIME;
	tSubStep1				:TIME;
	tSubStep2				:TIME;
	tSubStep3				:TIME;
	tSubStep4				:TIME;
	tSubStep5				:TIME;
	tSubStep6				:TIME;
	tSubStep7				:TIME;
	
	tSubStep1pt				:TIME;
	tSubStep2pt				:TIME;
	tSubStep3pt				:TIME;
	tSubStep4pt				:TIME;
	tSubStep5pt				:TIME;
	tSubStep6pt				:TIME;
	tSubStep7pt				:TIME;
	
	
	bHoldBar1				:BOOL;
	bHoldBar2				:BOOL;
	bHoldBar3				:BOOL;
	bHoldBar4				:BOOL;
	bHoldBar5				:BOOL;
	bHoldBar6				:BOOL;
	bHoldBar7				:BOOL;
	
	
	iCurrProc				:INT;
	

END_VAR
VAR // added by the converter: edge detectors and wires of the graphical bodies
    _w1, _w2, _w3, _w4, _w5, _w6, _w7, _w8, _w9, _w10, _w11, _w12, _w13, _w14, _w15 : TIME;
    _w16 : BOOL;
END_VAR

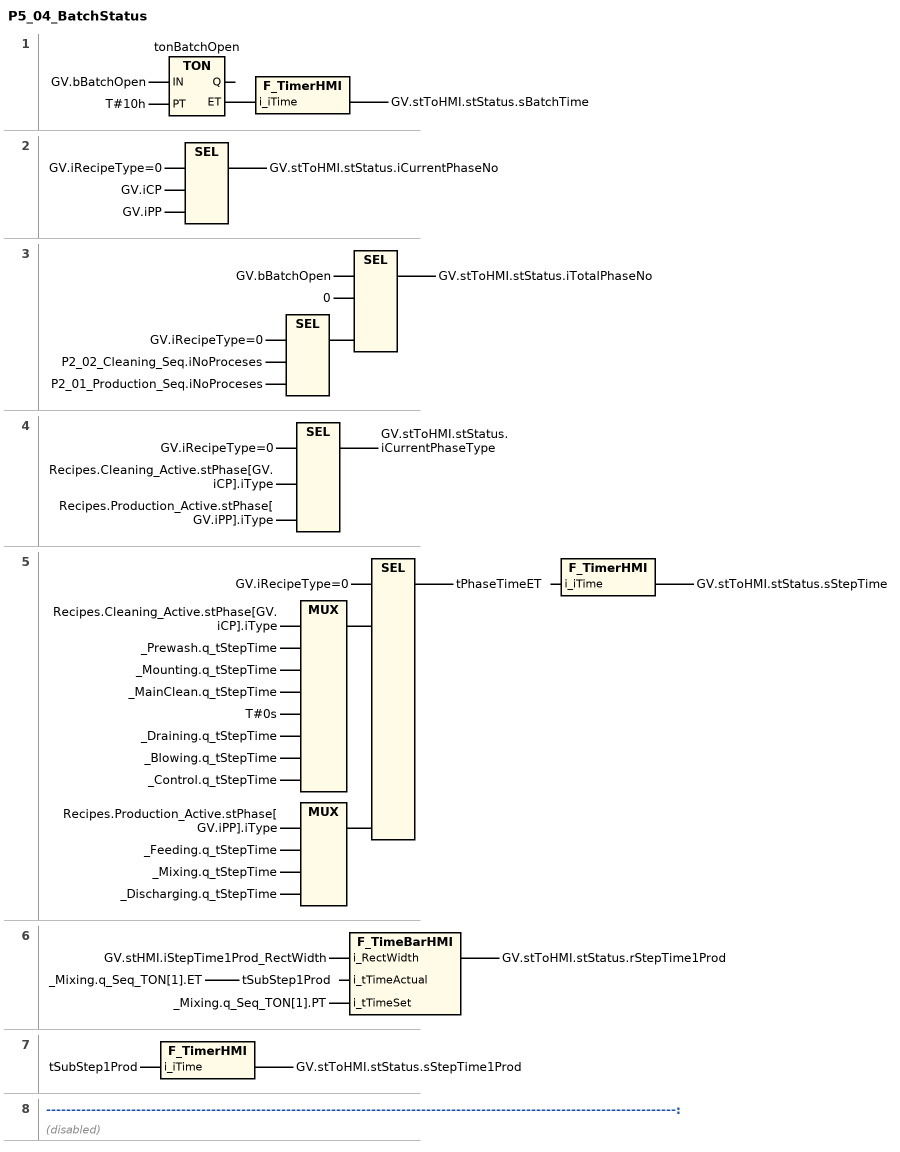
// NETWORK 1
tonBatchOpen(IN := GV.bBatchOpen, PT := T#10h); // TON
GV.stToHMI.stStatus.sBatchTime := F_TimerHMI(i_iTime := tonBatchOpen.ET);

// NETWORK 2
GV.stToHMI.stStatus.iCurrentPhaseNo := SEL(GV.iRecipeType=0, GV.iCP, GV.iPP);

// NETWORK 3
GV.stToHMI.stStatus.iTotalPhaseNo := SEL(GV.bBatchOpen, 0, SEL(GV.iRecipeType=0, P2_02_Cleaning_Seq.iNoProceses, P2_01_Production_Seq.iNoProceses));

// NETWORK 4
GV.stToHMI.stStatus.iCurrentPhaseType := SEL(GV.iRecipeType=0, Recipes.Cleaning_Active.stPhase[GV.iCP].iType, Recipes.Production_Active.stPhase[GV.iPP].iType);

// NETWORK 5
_w1 := SEL(GV.iRecipeType=0, MUX(Recipes.Cleaning_Active.stPhase[GV.iCP].iType, _Prewash.q_tStepTime, _Mounting.q_tStepTime, _MainClean.q_tStepTime, T#0s, _Draining.q_tStepTime, _Blowing.q_tStepTime, _Control.q_tStepTime), MUX(Recipes.Production_Active.stPhase[GV.iPP].iType, _Feeding.q_tStepTime, _Mixing.q_tStepTime, _Discharging.q_tStepTime));
tPhaseTimeET := _w1;
GV.stToHMI.stStatus.sStepTime := F_TimerHMI(i_iTime := _w1);

// NETWORK 6
tSubStep1Prod := _Mixing.q_Seq_TON[1].ET;
GV.stToHMI.stStatus.rStepTime1Prod := F_TimeBarHMI(i_RectWidth := GV.stHMI.iStepTime1Prod_RectWidth, i_tTimeActual := _Mixing.q_Seq_TON[1].ET, i_tTimeSet := _Mixing.q_Seq_TON[1].PT);

// NETWORK 7
GV.stToHMI.stStatus.sStepTime1Prod := F_TimerHMI(i_iTime := tSubStep1Prod);

// NETWORK 8 (disabled)
// label: ------------------------------------------------------------------------------------------------------------------------------

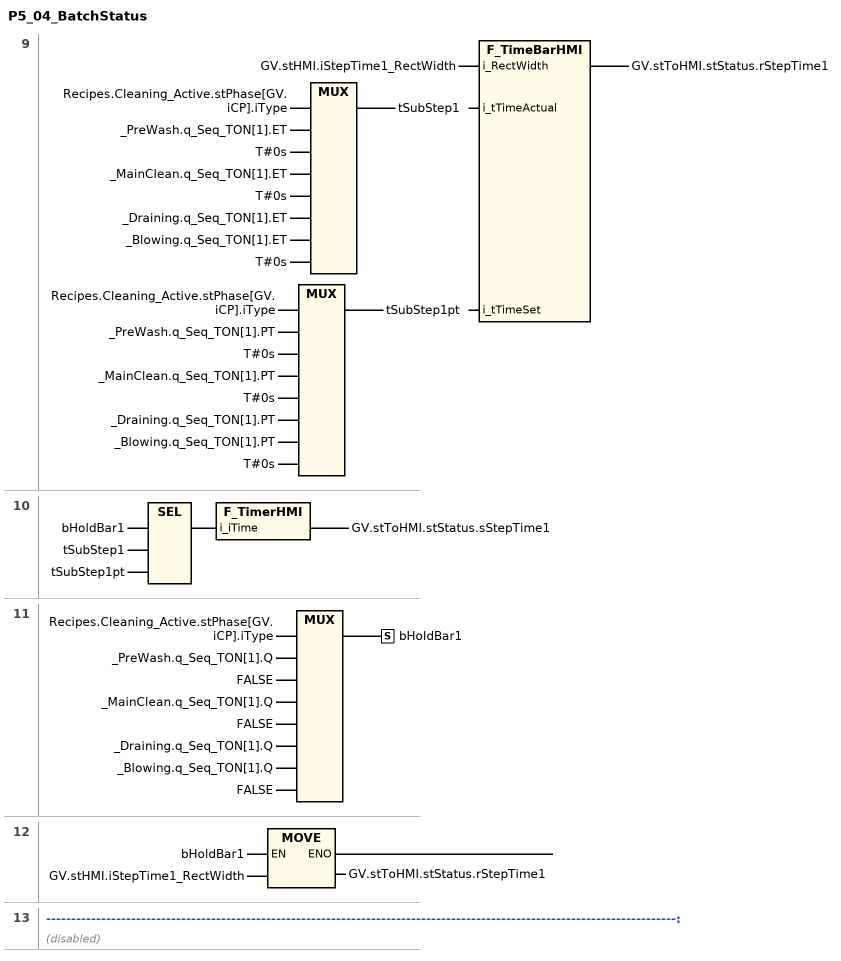
// NETWORK 9
_w2 := MUX(Recipes.Cleaning_Active.stPhase[GV.iCP].iType, _PreWash.q_Seq_TON[1].ET, T#0s, _MainClean.q_Seq_TON[1].ET, T#0s, _Draining.q_Seq_TON[1].ET, _Blowing.q_Seq_TON[1].ET, T#0s);
tSubStep1 := _w2;
_w3 := MUX(Recipes.Cleaning_Active.stPhase[GV.iCP].iType, _PreWash.q_Seq_TON[1].PT, T#0s, _MainClean.q_Seq_TON[1].PT, T#0s, _Draining.q_Seq_TON[1].PT, _Blowing.q_Seq_TON[1].PT, T#0s);
tSubStep1pt := _w3;
GV.stToHMI.stStatus.rStepTime1 := F_TimeBarHMI(i_RectWidth := GV.stHMI.iStepTime1_RectWidth, i_tTimeActual := _w2, i_tTimeSet := _w3);

// NETWORK 10
GV.stToHMI.stStatus.sStepTime1 := F_TimerHMI(i_iTime := SEL(bHoldBar1, tSubStep1, tSubStep1pt));

// NETWORK 11
bHoldBar1 S= MUX(Recipes.Cleaning_Active.stPhase[GV.iCP].iType, _PreWash.q_Seq_TON[1].Q, FALSE, _MainClean.q_Seq_TON[1].Q, FALSE, _Draining.q_Seq_TON[1].Q, _Blowing.q_Seq_TON[1].Q, FALSE);

// NETWORK 12
IF bHoldBar1 THEN GV.stToHMI.stStatus.rStepTime1 := GV.stHMI.iStepTime1_RectWidth; END_IF

// NETWORK 13 (disabled)
// label: ------------------------------------------------------------------------------------------------------------------------------

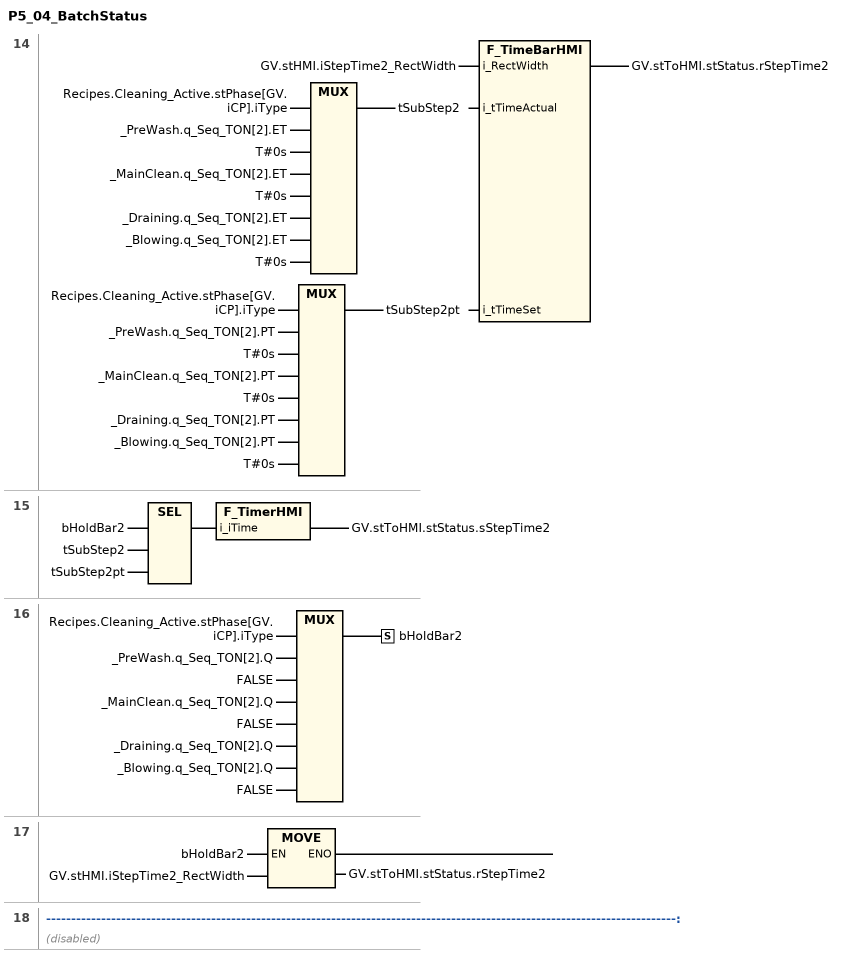
// NETWORK 14
_w4 := MUX(Recipes.Cleaning_Active.stPhase[GV.iCP].iType, _PreWash.q_Seq_TON[2].ET, T#0s, _MainClean.q_Seq_TON[2].ET, T#0s, _Draining.q_Seq_TON[2].ET, _Blowing.q_Seq_TON[2].ET, T#0s);
tSubStep2 := _w4;
_w5 := MUX(Recipes.Cleaning_Active.stPhase[GV.iCP].iType, _PreWash.q_Seq_TON[2].PT, T#0s, _MainClean.q_Seq_TON[2].PT, T#0s, _Draining.q_Seq_TON[2].PT, _Blowing.q_Seq_TON[2].PT, T#0s);
tSubStep2pt := _w5;
GV.stToHMI.stStatus.rStepTime2 := F_TimeBarHMI(i_RectWidth := GV.stHMI.iStepTime2_RectWidth, i_tTimeActual := _w4, i_tTimeSet := _w5);

// NETWORK 15
GV.stToHMI.stStatus.sStepTime2 := F_TimerHMI(i_iTime := SEL(bHoldBar2, tSubStep2, tSubStep2pt));

// NETWORK 16
bHoldBar2 S= MUX(Recipes.Cleaning_Active.stPhase[GV.iCP].iType, _PreWash.q_Seq_TON[2].Q, FALSE, _MainClean.q_Seq_TON[2].Q, FALSE, _Draining.q_Seq_TON[2].Q, _Blowing.q_Seq_TON[2].Q, FALSE);

// NETWORK 17
IF bHoldBar2 THEN GV.stToHMI.stStatus.rStepTime2 := GV.stHMI.iStepTime2_RectWidth; END_IF

// NETWORK 18 (disabled)
// label: ------------------------------------------------------------------------------------------------------------------------------

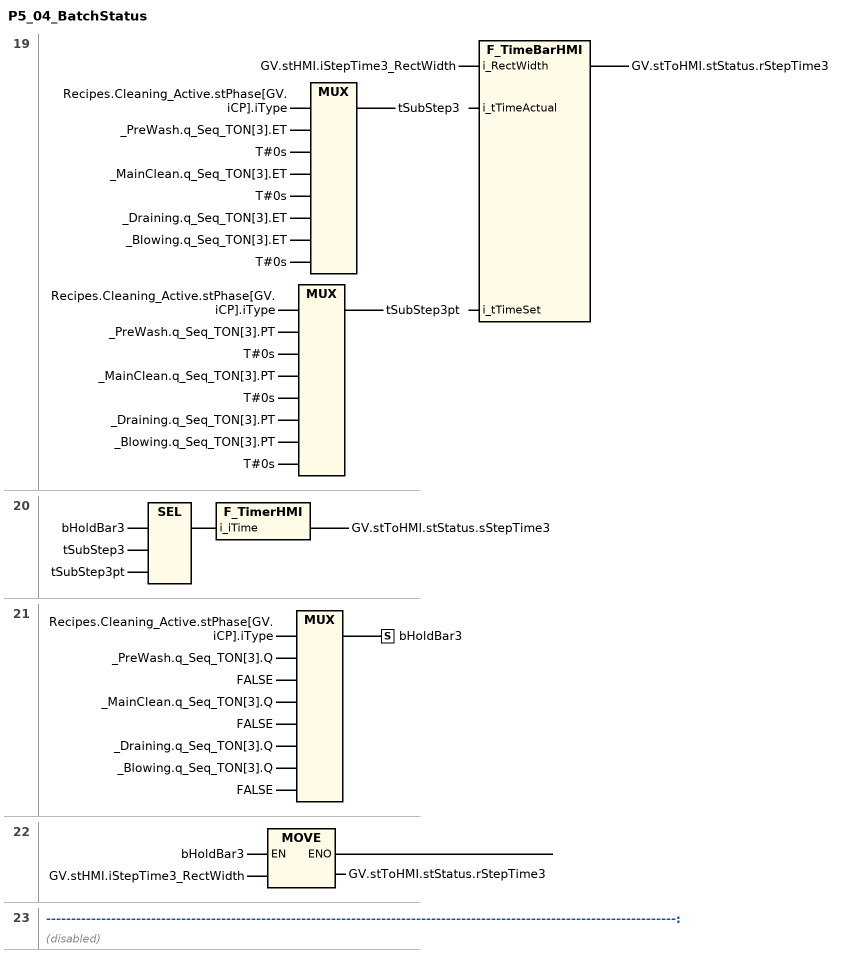
// NETWORK 19
_w6 := MUX(Recipes.Cleaning_Active.stPhase[GV.iCP].iType, _PreWash.q_Seq_TON[3].ET, T#0s, _MainClean.q_Seq_TON[3].ET, T#0s, _Draining.q_Seq_TON[3].ET, _Blowing.q_Seq_TON[3].ET, T#0s);
tSubStep3 := _w6;
_w7 := MUX(Recipes.Cleaning_Active.stPhase[GV.iCP].iType, _PreWash.q_Seq_TON[3].PT, T#0s, _MainClean.q_Seq_TON[3].PT, T#0s, _Draining.q_Seq_TON[3].PT, _Blowing.q_Seq_TON[3].PT, T#0s);
tSubStep3pt := _w7;
GV.stToHMI.stStatus.rStepTime3 := F_TimeBarHMI(i_RectWidth := GV.stHMI.iStepTime3_RectWidth, i_tTimeActual := _w6, i_tTimeSet := _w7);

// NETWORK 20
GV.stToHMI.stStatus.sStepTime3 := F_TimerHMI(i_iTime := SEL(bHoldBar3, tSubStep3, tSubStep3pt));

// NETWORK 21
bHoldBar3 S= MUX(Recipes.Cleaning_Active.stPhase[GV.iCP].iType, _PreWash.q_Seq_TON[3].Q, FALSE, _MainClean.q_Seq_TON[3].Q, FALSE, _Draining.q_Seq_TON[3].Q, _Blowing.q_Seq_TON[3].Q, FALSE);

// NETWORK 22
IF bHoldBar3 THEN GV.stToHMI.stStatus.rStepTime3 := GV.stHMI.iStepTime3_RectWidth; END_IF

// NETWORK 23 (disabled)
// label: ------------------------------------------------------------------------------------------------------------------------------

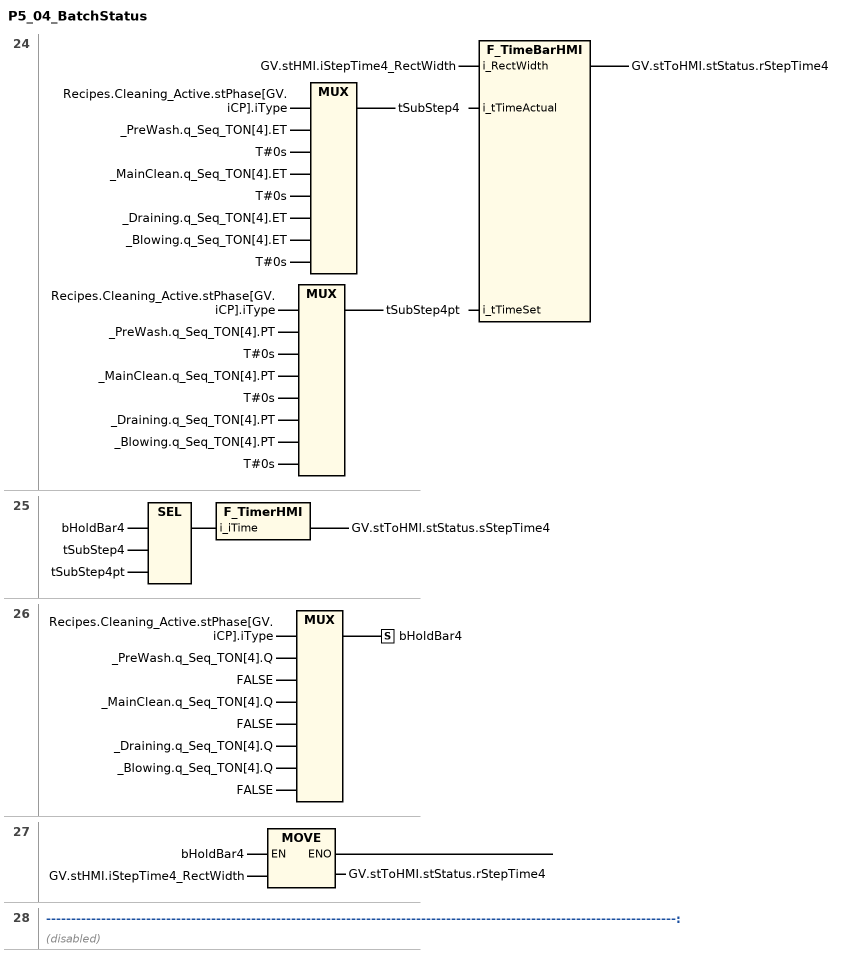
// NETWORK 24
_w8 := MUX(Recipes.Cleaning_Active.stPhase[GV.iCP].iType, _PreWash.q_Seq_TON[4].ET, T#0s, _MainClean.q_Seq_TON[4].ET, T#0s, _Draining.q_Seq_TON[4].ET, _Blowing.q_Seq_TON[4].ET, T#0s);
tSubStep4 := _w8;
_w9 := MUX(Recipes.Cleaning_Active.stPhase[GV.iCP].iType, _PreWash.q_Seq_TON[4].PT, T#0s, _MainClean.q_Seq_TON[4].PT, T#0s, _Draining.q_Seq_TON[4].PT, _Blowing.q_Seq_TON[4].PT, T#0s);
tSubStep4pt := _w9;
GV.stToHMI.stStatus.rStepTime4 := F_TimeBarHMI(i_RectWidth := GV.stHMI.iStepTime4_RectWidth, i_tTimeActual := _w8, i_tTimeSet := _w9);

// NETWORK 25
GV.stToHMI.stStatus.sStepTime4 := F_TimerHMI(i_iTime := SEL(bHoldBar4, tSubStep4, tSubStep4pt));

// NETWORK 26
bHoldBar4 S= MUX(Recipes.Cleaning_Active.stPhase[GV.iCP].iType, _PreWash.q_Seq_TON[4].Q, FALSE, _MainClean.q_Seq_TON[4].Q, FALSE, _Draining.q_Seq_TON[4].Q, _Blowing.q_Seq_TON[4].Q, FALSE);

// NETWORK 27
IF bHoldBar4 THEN GV.stToHMI.stStatus.rStepTime4 := GV.stHMI.iStepTime4_RectWidth; END_IF

// NETWORK 28 (disabled)
// label: ------------------------------------------------------------------------------------------------------------------------------

